{attribute 'qualified_only'}
{attribute 'strict'}
TYPE E_CX_NVXMLState : (
	IDLE,
	READXML,
	RESTORE,
	MONITOR,
	WRITEXML,
	BACKUP,
	RETRY
);
END_TYPE

(* stored: Version 1.1.0.1
   DUT E_CX_NVXMLState: Id {b20690d5-fb52-4d95-98d5-54c551d197b4} *)
